% RSLogix 500 project PROYECTO.RSS, saved by version 8.30.01.01 %
PROJECT "UNTITLED"    % processor: MicroLogix 1200 %

PROGRAM FILES
  LAD 2   21 rungs

DATA FILES
  O0 OUTPUT  4 elements
  I1 INPUT  4 elements
  S2 STATUS  66 elements
  B3 BINARY  1 elements
  T4 TIMER  1 elements
  C5 COUNTER  1 elements
  R6 CONTROL  1 elements
  N7 INTEGER  1 elements
  F8 FLOAT  1 elements

LADDER 2
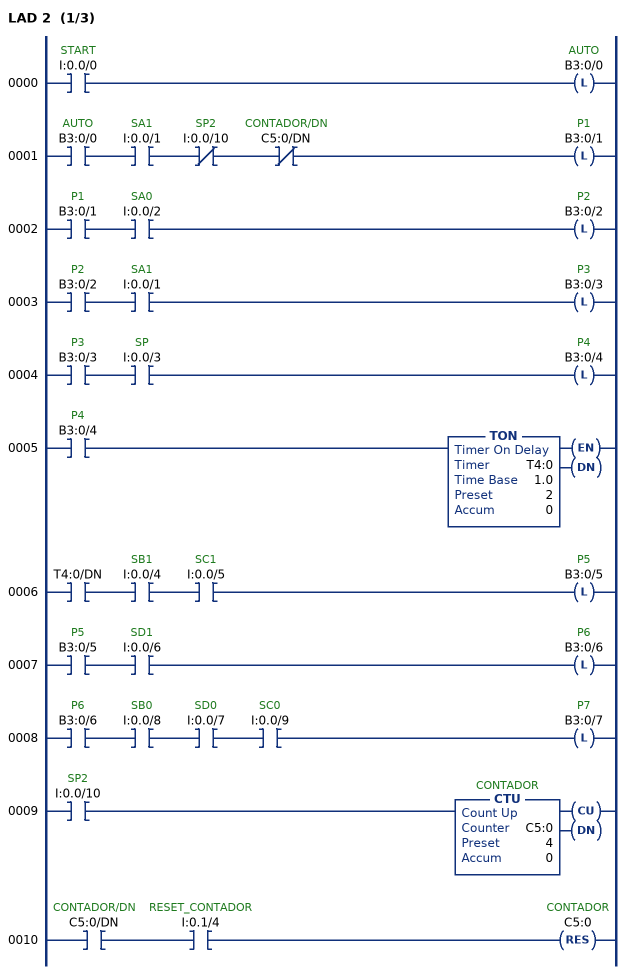
% Rung: 0 %
SOR XIC I:0.0/0 OTL B3:0/0 EOR
%   I:0.0/0  START %
%   B3:0/0  AUTO %
% Rung: 1 %
SOR XIC B3:0/0 XIC I:0.0/1 XIO I:0.0/10 XIO C5:0/DN OTL B3:0/1 EOR
%   B3:0/0  AUTO %
%   I:0.0/1  SA1 %
%   I:0.0/10  SP2 %
%   C5:0  CONTADOR %
%   B3:0/1  P1 %
% Rung: 2 %
SOR XIC B3:0/1 XIC I:0.0/2 OTL B3:0/2 EOR
%   B3:0/1  P1 %
%   I:0.0/2  SA0 %
%   B3:0/2  P2 %
% Rung: 3 %
SOR XIC B3:0/2 XIC I:0.0/1 OTL B3:0/3 EOR
%   B3:0/2  P2 %
%   I:0.0/1  SA1 %
%   B3:0/3  P3 %
% Rung: 4 %
SOR XIC B3:0/3 XIC I:0.0/3 OTL B3:0/4 EOR
%   B3:0/3  P3 %
%   I:0.0/3  SP %
%   B3:0/4  P4 %
% Rung: 5 %
SOR XIC B3:0/4 TON T4:0 1.0 2 0 EOR
%   B3:0/4  P4 %
% Rung: 6 %
SOR XIC T4:0/DN XIC I:0.0/4 XIC I:0.0/5 OTL B3:0/5 EOR
%   I:0.0/4  SB1 %
%   I:0.0/5  SC1 %
%   B3:0/5  P5 %
% Rung: 7 %
SOR XIC B3:0/5 XIC I:0.0/6 OTL B3:0/6 EOR
%   B3:0/5  P5 %
%   I:0.0/6  SD1 %
%   B3:0/6  P6 %
% Rung: 8 %
SOR XIC B3:0/6 XIC I:0.0/8 XIC I:0.0/7 XIC I:0.0/9 OTL B3:0/7 EOR
%   B3:0/6  P6 %
%   I:0.0/8  SB0 %
%   I:0.0/7  SD0 %
%   I:0.0/9  SC0 %
%   B3:0/7  P7 %
% Rung: 9 %
SOR XIC I:0.0/10 CTU C5:0 4 0 EOR
%   I:0.0/10  SP2 %
%   C5:0  CONTADOR %
% Rung: 10 %
SOR XIC C5:0/DN XIC I:0.1/4 RES C5:0 EOR
%   C5:0  CONTADOR %
%   I:0.1/4  RESET_CONTADOR %

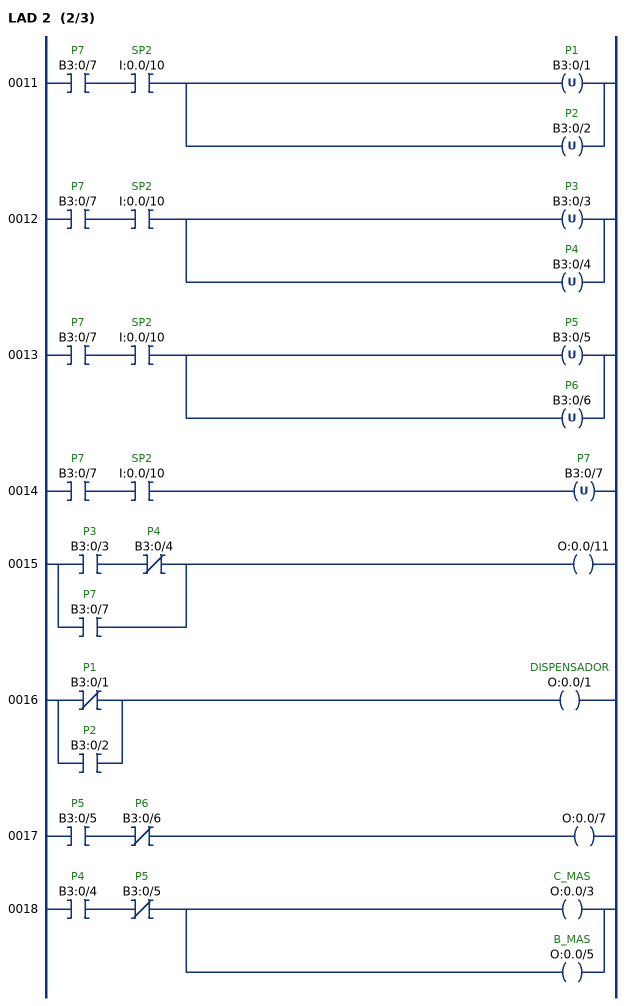
% Rung: 11 %
SOR XIC B3:0/7 XIC I:0.0/10 BST OTU B3:0/1 NXB OTU B3:0/2 BND EOR
%   B3:0/7  P7 %
%   I:0.0/10  SP2 %
%   B3:0/1  P1 %
%   B3:0/2  P2 %
% Rung: 12 %
SOR XIC B3:0/7 XIC I:0.0/10 BST OTU B3:0/3 NXB OTU B3:0/4 BND EOR
%   B3:0/7  P7 %
%   I:0.0/10  SP2 %
%   B3:0/3  P3 %
%   B3:0/4  P4 %
% Rung: 13 %
SOR XIC B3:0/7 XIC I:0.0/10 BST OTU B3:0/5 NXB OTU B3:0/6 BND EOR
%   B3:0/7  P7 %
%   I:0.0/10  SP2 %
%   B3:0/5  P5 %
%   B3:0/6  P6 %
% Rung: 14 %
SOR XIC B3:0/7 XIC I:0.0/10 OTU B3:0/7 EOR
%   B3:0/7  P7 %
%   I:0.0/10  SP2 %
% Rung: 15 %
SOR BST XIC B3:0/3 XIO B3:0/4 NXB XIC B3:0/7 BND OTE O:0.0/11 EOR
%   B3:0/3  P3 %
%   B3:0/4  P4 %
%   B3:0/7  P7 %
% Rung: 16 %
SOR BST XIO B3:0/1 NXB XIC B3:0/2 BND OTE O:0.0/1 EOR
%   B3:0/1  P1 %
%   B3:0/2  P2 %
%   O:0.0/1  DISPENSADOR %
% Rung: 17 %
SOR XIC B3:0/5 XIO B3:0/6 OTE O:0.0/7 EOR
%   B3:0/5  P5 %
%   B3:0/6  P6 %
% Rung: 18 %
SOR XIC B3:0/4 XIO B3:0/5 BST OTE O:0.0/3 NXB OTE O:0.0/5 BND EOR
%   B3:0/4  P4 %
%   B3:0/5  P5 %
%   O:0.0/3  C_MAS %
%   O:0.0/5  B_MAS %

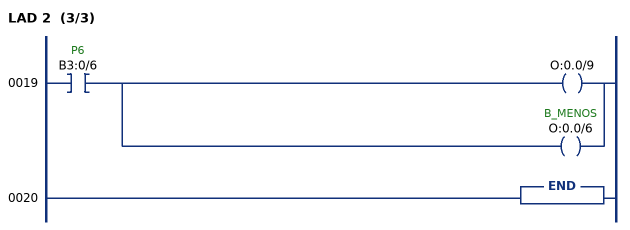
% Rung: 19 %
SOR XIC B3:0/6 BST OTE O:0.0/9 NXB OTE O:0.0/6 BND EOR
%   B3:0/6  P6 %
%   O:0.0/6  B_MENOS %
% Rung: 20 %
SOR END EOR

OTHER DOCUMENTED ADDRESSES
  O:0.0/0  MOTOR
  O:0.0/2  ESTAMPADOR
  O:0.0/4  C_MENOS

DATA TABLE (non-zero values as saved)
DATA T4
% .PRE .ACC %
% T4:0 % 2 0
DATA C5
% .PRE .ACC %
% C5:0 % 4 0
